ABB RAPID module: Module1.modx

MODULE Module1
    CONST robtarget Target_10:=[[355.425625842,0,585],[0.5,0,0.866025404,0],[0,0,0,0],[9E+09,9E+09,9E+09,9E+09,9E+09,9E+09]];
    CONST robtarget Target_20:=[[210.419326539,-286.445601335,585],[0.44609706,0.391142223,0.772662773,-0.225826068],[-1,-1,-1,0],[9E+09,9E+09,9E+09,9E+09,9E+09,9E+09]];

    CONST jointtarget JointTarget_0:=[[179.42,0.01,0.61,-29.68,-1.17,209.68],[9E+09,9E+09,9E+09,9E+09,9E+09,9E+09]];
    CONST jointtarget JointTarget_1:=[[178.84,0.03,1.21,-35.31,-2.01,215.3],[9E+09,9E+09,9E+09,9E+09,9E+09,9E+09]];
    CONST jointtarget JointTarget_2:=[[178.26,0.07,1.79,-37.62,-2.86,217.6],[9E+09,9E+09,9E+09,9E+09,9E+09,9E+09]];
    CONST jointtarget JointTarget_3:=[[177.68,0.12,2.37,-38.88,-3.7,218.83],[9E+09,9E+09,9E+09,9E+09,9E+09,9E+09]];
    CONST jointtarget JointTarget_4:=[[177.1,0.18,2.92,-39.66,-4.55,219.59],[9E+09,9E+09,9E+09,9E+09,9E+09,9E+09]];
    CONST jointtarget JointTarget_5:=[[176.52,0.26,3.47,-40.2,-5.4,220.1],[9E+09,9E+09,9E+09,9E+09,9E+09,9E+09]];
    CONST jointtarget JointTarget_6:=[[175.94,0.35,4.01,-40.6,-6.24,220.46],[9E+09,9E+09,9E+09,9E+09,9E+09,9E+09]];
    CONST jointtarget JointTarget_7:=[[175.36,0.45,4.53,-40.9,-7.09,220.71],[9E+09,9E+09,9E+09,9E+09,9E+09,9E+09]];
    CONST jointtarget JointTarget_8:=[[174.79,0.56,5.03,-41.13,-7.94,220.9],[9E+09,9E+09,9E+09,9E+09,9E+09,9E+09]];
    CONST jointtarget JointTarget_9:=[[174.21,0.69,5.53,-41.33,-8.78,221.03],[9E+09,9E+09,9E+09,9E+09,9E+09,9E+09]];
    CONST jointtarget JointTarget_10:=[[173.64,0.83,6.01,-41.49,-9.63,221.13],[9E+09,9E+09,9E+09,9E+09,9E+09,9E+09]];
    CONST jointtarget JointTarget_11:=[[173.07,0.98,6.48,-41.62,-10.47,221.19],[9E+09,9E+09,9E+09,9E+09,9E+09,9E+09]];
    CONST jointtarget JointTarget_12:=[[172.49,1.15,6.94,-41.74,-11.31,221.24],[9E+09,9E+09,9E+09,9E+09,9E+09,9E+09]];
    CONST jointtarget JointTarget_13:=[[171.93,1.33,7.38,-41.84,-12.15,221.26],[9E+09,9E+09,9E+09,9E+09,9E+09,9E+09]];
    CONST jointtarget JointTarget_14:=[[171.36,1.52,7.82,-41.94,-12.99,221.26],[9E+09,9E+09,9E+09,9E+09,9E+09,9E+09]];
    CONST jointtarget JointTarget_15:=[[170.79,1.73,8.23,-42.02,-13.83,221.25],[9E+09,9E+09,9E+09,9E+09,9E+09,9E+09]];
    CONST jointtarget JointTarget_16:=[[170.23,1.94,8.64,-42.1,-14.67,221.22],[9E+09,9E+09,9E+09,9E+09,9E+09,9E+09]];
    CONST jointtarget JointTarget_17:=[[169.67,2.17,9.03,-42.17,-15.5,221.19],[9E+09,9E+09,9E+09,9E+09,9E+09,9E+09]];
    CONST jointtarget JointTarget_18:=[[169.11,2.42,9.42,-42.24,-16.33,221.14],[9E+09,9E+09,9E+09,9E+09,9E+09,9E+09]];
    CONST jointtarget JointTarget_19:=[[168.55,2.67,9.78,-42.3,-17.16,221.09],[9E+09,9E+09,9E+09,9E+09,9E+09,9E+09]];
    CONST jointtarget JointTarget_20:=[[167.99,2.94,10.14,-42.36,-17.99,221.02],[9E+09,9E+09,9E+09,9E+09,9E+09,9E+09]];
    CONST jointtarget JointTarget_21:=[[167.44,3.22,10.48,-42.42,-18.81,220.95],[9E+09,9E+09,9E+09,9E+09,9E+09,9E+09]];
    CONST jointtarget JointTarget_22:=[[166.89,3.52,10.81,-42.48,-19.63,220.87],[9E+09,9E+09,9E+09,9E+09,9E+09,9E+09]];
    CONST jointtarget JointTarget_23:=[[166.34,3.82,11.13,-42.54,-20.45,220.78],[9E+09,9E+09,9E+09,9E+09,9E+09,9E+09]];
    CONST jointtarget JointTarget_24:=[[165.79,4.14,11.43,-42.6,-21.26,220.69],[9E+09,9E+09,9E+09,9E+09,9E+09,9E+09]];
    CONST jointtarget JointTarget_25:=[[165.25,4.47,11.72,-42.65,-22.07,220.6],[9E+09,9E+09,9E+09,9E+09,9E+09,9E+09]];
    CONST jointtarget JointTarget_26:=[[164.71,4.82,12,-42.71,-22.88,220.49],[9E+09,9E+09,9E+09,9E+09,9E+09,9E+09]];
    CONST jointtarget JointTarget_27:=[[164.17,5.17,12.26,-42.77,-23.68,220.38],[9E+09,9E+09,9E+09,9E+09,9E+09,9E+09]];
    CONST jointtarget JointTarget_28:=[[163.64,5.54,12.51,-42.83,-24.48,220.27],[9E+09,9E+09,9E+09,9E+09,9E+09,9E+09]];
    CONST jointtarget JointTarget_29:=[[163.11,5.91,12.75,-42.89,-25.27,220.16],[9E+09,9E+09,9E+09,9E+09,9E+09,9E+09]];
    CONST jointtarget JointTarget_30:=[[162.58,6.3,12.97,-42.96,-26.06,220.03],[9E+09,9E+09,9E+09,9E+09,9E+09,9E+09]];
    CONST jointtarget JointTarget_31:=[[162.05,6.7,13.19,-43.02,-26.85,219.91],[9E+09,9E+09,9E+09,9E+09,9E+09,9E+09]];
    CONST jointtarget JointTarget_32:=[[161.53,7.12,13.38,-43.09,-27.63,219.78],[9E+09,9E+09,9E+09,9E+09,9E+09,9E+09]];
    CONST jointtarget JointTarget_33:=[[161.01,7.54,13.57,-43.16,-28.41,219.65],[9E+09,9E+09,9E+09,9E+09,9E+09,9E+09]];
    CONST jointtarget JointTarget_34:=[[160.49,7.97,13.74,-43.23,-29.18,219.52],[9E+09,9E+09,9E+09,9E+09,9E+09,9E+09]];
    CONST jointtarget JointTarget_35:=[[159.98,8.42,13.9,-43.3,-29.94,219.38],[9E+09,9E+09,9E+09,9E+09,9E+09,9E+09]];
    CONST jointtarget JointTarget_36:=[[159.47,8.88,14.04,-43.37,-30.7,219.24],[9E+09,9E+09,9E+09,9E+09,9E+09,9E+09]];
    CONST jointtarget JointTarget_37:=[[158.97,9.34,14.18,-43.45,-31.46,219.1],[9E+09,9E+09,9E+09,9E+09,9E+09,9E+09]];
    CONST jointtarget JointTarget_38:=[[158.47,9.82,14.29,-43.53,-32.2,218.95],[9E+09,9E+09,9E+09,9E+09,9E+09,9E+09]];
    CONST jointtarget JointTarget_39:=[[157.97,10.31,14.4,-43.61,-32.94,218.81],[9E+09,9E+09,9E+09,9E+09,9E+09,9E+09]];
    CONST jointtarget JointTarget_40:=[[157.47,10.8,14.49,-43.7,-33.68,218.66],[9E+09,9E+09,9E+09,9E+09,9E+09,9E+09]];
    CONST jointtarget JointTarget_41:=[[156.98,11.31,14.57,-43.79,-34.41,218.51],[9E+09,9E+09,9E+09,9E+09,9E+09,9E+09]];
    CONST jointtarget JointTarget_42:=[[156.49,11.83,14.63,-43.88,-35.13,218.36],[9E+09,9E+09,9E+09,9E+09,9E+09,9E+09]];
    CONST jointtarget JointTarget_43:=[[156.01,12.35,14.68,-43.97,-35.85,218.2],[9E+09,9E+09,9E+09,9E+09,9E+09,9E+09]];
    CONST jointtarget JointTarget_44:=[[155.53,12.89,14.72,-44.07,-36.55,218.05],[9E+09,9E+09,9E+09,9E+09,9E+09,9E+09]];
    CONST jointtarget JointTarget_45:=[[155.05,13.43,14.74,-44.17,-37.25,217.9],[9E+09,9E+09,9E+09,9E+09,9E+09,9E+09]];
    CONST jointtarget JointTarget_46:=[[154.58,13.98,14.76,-44.27,-37.95,217.74],[9E+09,9E+09,9E+09,9E+09,9E+09,9E+09]];
    CONST jointtarget JointTarget_47:=[[154.11,14.54,14.75,-44.38,-38.63,217.59],[9E+09,9E+09,9E+09,9E+09,9E+09,9E+09]];
    CONST jointtarget JointTarget_48:=[[153.64,15.11,14.74,-44.49,-39.31,217.43],[9E+09,9E+09,9E+09,9E+09,9E+09,9E+09]];
    CONST jointtarget JointTarget_49:=[[153.18,15.69,14.71,-44.6,-39.98,217.28],[9E+09,9E+09,9E+09,9E+09,9E+09,9E+09]];
    CONST jointtarget JointTarget_50:=[[153.87,15.35,15.18,-43.63,-39.67,216.46],[9E+09,9E+09,9E+09,9E+09,9E+09,9E+09]];
    CONST jointtarget JointTarget_51:=[[154.56,15.02,15.64,-42.64,-39.35,215.64],[9E+09,9E+09,9E+09,9E+09,9E+09,9E+09]];
    CONST jointtarget JointTarget_52:=[[155.26,14.7,16.09,-41.63,-39.04,214.8],[9E+09,9E+09,9E+09,9E+09,9E+09,9E+09]];
    CONST jointtarget JointTarget_53:=[[155.98,14.38,16.52,-40.59,-38.73,213.94],[9E+09,9E+09,9E+09,9E+09,9E+09,9E+09]];
    CONST jointtarget JointTarget_54:=[[156.69,14.08,16.94,-39.54,-38.42,213.06],[9E+09,9E+09,9E+09,9E+09,9E+09,9E+09]];
    CONST jointtarget JointTarget_55:=[[157.42,13.78,17.35,-38.46,-38.12,212.17],[9E+09,9E+09,9E+09,9E+09,9E+09,9E+09]];
    CONST jointtarget JointTarget_56:=[[158.16,13.5,17.74,-37.36,-37.82,211.26],[9E+09,9E+09,9E+09,9E+09,9E+09,9E+09]];
    CONST jointtarget JointTarget_57:=[[158.9,13.22,18.12,-36.24,-37.52,210.32],[9E+09,9E+09,9E+09,9E+09,9E+09,9E+09]];
    CONST jointtarget JointTarget_58:=[[159.65,12.95,18.49,-35.09,-37.23,209.37],[9E+09,9E+09,9E+09,9E+09,9E+09,9E+09]];
    CONST jointtarget JointTarget_59:=[[160.41,12.69,18.85,-33.92,-36.94,208.4],[9E+09,9E+09,9E+09,9E+09,9E+09,9E+09]];
    CONST jointtarget JointTarget_60:=[[161.17,12.45,19.19,-32.72,-36.66,207.4],[9E+09,9E+09,9E+09,9E+09,9E+09,9E+09]];
    CONST jointtarget JointTarget_61:=[[161.94,12.21,19.52,-31.5,-36.39,206.39],[9E+09,9E+09,9E+09,9E+09,9E+09,9E+09]];
    CONST jointtarget JointTarget_62:=[[162.72,11.98,19.83,-30.26,-36.12,205.36],[9E+09,9E+09,9E+09,9E+09,9E+09,9E+09]];
    CONST jointtarget JointTarget_63:=[[163.5,11.76,20.13,-28.99,-35.86,204.3],[9E+09,9E+09,9E+09,9E+09,9E+09,9E+09]];
    CONST jointtarget JointTarget_64:=[[164.29,11.55,20.42,-27.7,-35.62,203.22],[9E+09,9E+09,9E+09,9E+09,9E+09,9E+09]];
    CONST jointtarget JointTarget_65:=[[165.09,11.36,20.69,-26.38,-35.38,202.13],[9E+09,9E+09,9E+09,9E+09,9E+09,9E+09]];
    CONST jointtarget JointTarget_66:=[[165.9,11.17,20.95,-25.04,-35.15,201.01],[9E+09,9E+09,9E+09,9E+09,9E+09,9E+09]];
    CONST jointtarget JointTarget_67:=[[166.7,11,21.19,-23.68,-34.93,199.87],[9E+09,9E+09,9E+09,9E+09,9E+09,9E+09]];
    CONST jointtarget JointTarget_68:=[[167.52,10.83,21.43,-22.3,-34.72,198.72],[9E+09,9E+09,9E+09,9E+09,9E+09,9E+09]];
    CONST jointtarget JointTarget_69:=[[168.34,10.68,21.64,-20.89,-34.53,197.54],[9E+09,9E+09,9E+09,9E+09,9E+09,9E+09]];
    CONST jointtarget JointTarget_70:=[[169.16,10.54,21.85,-19.47,-34.34,196.35],[9E+09,9E+09,9E+09,9E+09,9E+09,9E+09]];
    CONST jointtarget JointTarget_71:=[[169.99,10.41,22.04,-18.02,-34.17,195.14],[9E+09,9E+09,9E+09,9E+09,9E+09,9E+09]];
    CONST jointtarget JointTarget_72:=[[170.83,10.29,22.21,-16.56,-34.02,193.91],[9E+09,9E+09,9E+09,9E+09,9E+09,9E+09]];
    CONST jointtarget JointTarget_73:=[[171.66,10.18,22.37,-15.08,-33.88,192.67],[9E+09,9E+09,9E+09,9E+09,9E+09,9E+09]];
    CONST jointtarget JointTarget_74:=[[172.5,10.08,22.52,-13.58,-33.75,191.41],[9E+09,9E+09,9E+09,9E+09,9E+09,9E+09]];
    CONST jointtarget JointTarget_75:=[[173.35,10,22.65,-12.07,-33.64,190.14],[9E+09,9E+09,9E+09,9E+09,9E+09,9E+09]];
    CONST jointtarget JointTarget_76:=[[174.19,9.93,22.77,-10.55,-33.55,188.86],[9E+09,9E+09,9E+09,9E+09,9E+09,9E+09]];
    CONST jointtarget JointTarget_77:=[[175.04,9.87,22.87,-9.01,-33.47,187.57],[9E+09,9E+09,9E+09,9E+09,9E+09,9E+09]];
    CONST jointtarget JointTarget_78:=[[175.9,9.82,22.96,-7.47,-33.41,186.27],[9E+09,9E+09,9E+09,9E+09,9E+09,9E+09]];
    CONST jointtarget JointTarget_79:=[[176.75,9.79,23.04,-5.92,-33.36,184.97],[9E+09,9E+09,9E+09,9E+09,9E+09,9E+09]];
    CONST jointtarget JointTarget_80:=[[177.6,9.76,23.1,-4.36,-33.33,183.66],[9E+09,9E+09,9E+09,9E+09,9E+09,9E+09]];
    CONST jointtarget JointTarget_81:=[[178.46,9.75,23.14,-2.8,-33.32,182.35],[9E+09,9E+09,9E+09,9E+09,9E+09,9E+09]];
    CONST jointtarget JointTarget_82:=[[179.32,9.75,23.17,-1.24,-33.33,181.04],[9E+09,9E+09,9E+09,9E+09,9E+09,9E+09]];
    CONST jointtarget JointTarget_83:=[[180.17,9.76,23.19,0.32,-33.35,179.73],[9E+09,9E+09,9E+09,9E+09,9E+09,9E+09]];
    CONST jointtarget JointTarget_84:=[[181.03,9.79,23.19,1.87,-33.39,178.43],[9E+09,9E+09,9E+09,9E+09,9E+09,9E+09]];
    CONST jointtarget JointTarget_85:=[[181.89,9.83,23.18,3.43,-33.45,177.13],[9E+09,9E+09,9E+09,9E+09,9E+09,9E+09]];
    CONST jointtarget JointTarget_86:=[[182.74,9.88,23.15,4.97,-33.53,175.83],[9E+09,9E+09,9E+09,9E+09,9E+09,9E+09]];
    CONST jointtarget JointTarget_87:=[[183.6,9.94,23.11,6.51,-33.62,174.55],[9E+09,9E+09,9E+09,9E+09,9E+09,9E+09]];
    CONST jointtarget JointTarget_88:=[[184.45,10.01,23.06,8.03,-33.73,173.27],[9E+09,9E+09,9E+09,9E+09,9E+09,9E+09]];
    CONST jointtarget JointTarget_89:=[[185.3,10.1,22.98,9.55,-33.85,172.01],[9E+09,9E+09,9E+09,9E+09,9E+09,9E+09]];
    CONST jointtarget JointTarget_90:=[[186.15,10.19,22.9,11.05,-33.99,170.76],[9E+09,9E+09,9E+09,9E+09,9E+09,9E+09]];
    CONST jointtarget JointTarget_91:=[[187,10.3,22.8,12.53,-34.14,169.53],[9E+09,9E+09,9E+09,9E+09,9E+09,9E+09]];
    CONST jointtarget JointTarget_92:=[[187.84,10.42,22.69,14,-34.31,168.31],[9E+09,9E+09,9E+09,9E+09,9E+09,9E+09]];
    CONST jointtarget JointTarget_93:=[[188.68,10.55,22.56,15.45,-34.49,167.11],[9E+09,9E+09,9E+09,9E+09,9E+09,9E+09]];
    CONST jointtarget JointTarget_94:=[[189.51,10.7,22.42,16.88,-34.69,165.92],[9E+09,9E+09,9E+09,9E+09,9E+09,9E+09]];
    CONST jointtarget JointTarget_95:=[[190.34,10.85,22.26,18.29,-34.9,164.76],[9E+09,9E+09,9E+09,9E+09,9E+09,9E+09]];
    CONST jointtarget JointTarget_96:=[[191.17,11.02,22.09,19.68,-35.12,163.61],[9E+09,9E+09,9E+09,9E+09,9E+09,9E+09]];
    CONST jointtarget JointTarget_97:=[[191.99,11.2,21.9,21.05,-35.35,162.49],[9E+09,9E+09,9E+09,9E+09,9E+09,9E+09]];
    CONST jointtarget JointTarget_98:=[[192.81,11.39,21.7,22.39,-35.6,161.39],[9E+09,9E+09,9E+09,9E+09,9E+09,9E+09]];
    CONST jointtarget JointTarget_99:=[[193.62,11.59,21.49,23.71,-35.85,160.3],[9E+09,9E+09,9E+09,9E+09,9E+09,9E+09]];
    CONST jointtarget JointTarget_100:=[[193.15,11.97,21.97,22.48,-36.49,161.5],[9E+09,9E+09,9E+09,9E+09,9E+09,9E+09]];
    CONST jointtarget JointTarget_101:=[[192.67,12.37,22.44,21.3,-37.15,162.65],[9E+09,9E+09,9E+09,9E+09,9E+09,9E+09]];
    CONST jointtarget JointTarget_102:=[[192.19,12.79,22.89,20.15,-37.82,163.75],[9E+09,9E+09,9E+09,9E+09,9E+09,9E+09]];
    CONST jointtarget JointTarget_103:=[[191.71,13.22,23.33,19.03,-38.51,164.81],[9E+09,9E+09,9E+09,9E+09,9E+09,9E+09]];
    CONST jointtarget JointTarget_104:=[[191.23,13.67,23.75,17.95,-39.22,165.83],[9E+09,9E+09,9E+09,9E+09,9E+09,9E+09]];
    CONST jointtarget JointTarget_105:=[[190.75,14.14,24.15,16.9,-39.93,166.81],[9E+09,9E+09,9E+09,9E+09,9E+09,9E+09]];
    CONST jointtarget JointTarget_106:=[[190.27,14.62,24.54,15.88,-40.66,167.75],[9E+09,9E+09,9E+09,9E+09,9E+09,9E+09]];
    CONST jointtarget JointTarget_107:=[[189.78,15.12,24.91,14.89,-41.41,168.66],[9E+09,9E+09,9E+09,9E+09,9E+09,9E+09]];
    CONST jointtarget JointTarget_108:=[[189.3,15.64,25.26,13.93,-42.16,169.52],[9E+09,9E+09,9E+09,9E+09,9E+09,9E+09]];
    CONST jointtarget JointTarget_109:=[[188.81,16.18,25.6,12.99,-42.92,170.35],[9E+09,9E+09,9E+09,9E+09,9E+09,9E+09]];
    CONST jointtarget JointTarget_110:=[[188.32,16.73,25.92,12.09,-43.69,171.14],[9E+09,9E+09,9E+09,9E+09,9E+09,9E+09]];
    CONST jointtarget JointTarget_111:=[[187.83,17.3,26.22,11.21,-44.47,171.9],[9E+09,9E+09,9E+09,9E+09,9E+09,9E+09]];
    CONST jointtarget JointTarget_112:=[[187.34,17.88,26.51,10.36,-45.26,172.62],[9E+09,9E+09,9E+09,9E+09,9E+09,9E+09]];
    CONST jointtarget JointTarget_113:=[[186.84,18.48,26.78,9.53,-46.06,173.31],[9E+09,9E+09,9E+09,9E+09,9E+09,9E+09]];
    CONST jointtarget JointTarget_114:=[[186.35,19.09,27.03,8.72,-46.86,173.97],[9E+09,9E+09,9E+09,9E+09,9E+09,9E+09]];
    CONST jointtarget JointTarget_115:=[[185.86,19.72,27.27,7.93,-47.66,174.6],[9E+09,9E+09,9E+09,9E+09,9E+09,9E+09]];
    CONST jointtarget JointTarget_116:=[[185.36,20.37,27.48,7.17,-48.47,175.2],[9E+09,9E+09,9E+09,9E+09,9E+09,9E+09]];
    CONST jointtarget JointTarget_117:=[[184.86,21.02,27.68,6.42,-49.29,175.77],[9E+09,9E+09,9E+09,9E+09,9E+09,9E+09]];
    CONST jointtarget JointTarget_118:=[[184.37,21.7,27.87,5.7,-50.1,176.31],[9E+09,9E+09,9E+09,9E+09,9E+09,9E+09]];
    CONST jointtarget JointTarget_119:=[[183.87,22.38,28.03,4.99,-50.92,176.82],[9E+09,9E+09,9E+09,9E+09,9E+09,9E+09]];
    CONST jointtarget JointTarget_120:=[[183.37,23.09,28.18,4.29,-51.74,177.31],[9E+09,9E+09,9E+09,9E+09,9E+09,9E+09]];
    CONST jointtarget JointTarget_121:=[[182.87,23.8,28.3,3.62,-52.56,177.78],[9E+09,9E+09,9E+09,9E+09,9E+09,9E+09]];
    CONST jointtarget JointTarget_122:=[[182.37,24.53,28.41,2.96,-53.37,178.22],[9E+09,9E+09,9E+09,9E+09,9E+09,9E+09]];
    CONST jointtarget JointTarget_123:=[[181.87,25.26,28.5,2.31,-54.19,178.64],[9E+09,9E+09,9E+09,9E+09,9E+09,9E+09]];
    CONST jointtarget JointTarget_124:=[[181.37,26.02,28.58,1.68,-55,179.03],[9E+09,9E+09,9E+09,9E+09,9E+09,9E+09]];
    CONST jointtarget JointTarget_125:=[[180.87,26.78,28.63,1.05,-55.81,179.4],[9E+09,9E+09,9E+09,9E+09,9E+09,9E+09]];
    CONST jointtarget JointTarget_126:=[[180.37,27.55,28.67,0.45,-56.62,179.75],[9E+09,9E+09,9E+09,9E+09,9E+09,9E+09]];
    CONST jointtarget JointTarget_127:=[[179.87,28.33,28.69,-0.15,-57.42,180.08],[9E+09,9E+09,9E+09,9E+09,9E+09,9E+09]];
    CONST jointtarget JointTarget_128:=[[179.37,29.13,28.69,-0.74,-58.22,180.39],[9E+09,9E+09,9E+09,9E+09,9E+09,9E+09]];
    CONST jointtarget JointTarget_129:=[[178.87,29.93,28.67,-1.32,-59.01,180.69],[9E+09,9E+09,9E+09,9E+09,9E+09,9E+09]];
    CONST jointtarget JointTarget_130:=[[178.37,30.74,28.64,-1.89,-59.79,180.96],[9E+09,9E+09,9E+09,9E+09,9E+09,9E+09]];
    CONST jointtarget JointTarget_131:=[[177.87,31.56,28.58,-2.44,-60.57,181.22],[9E+09,9E+09,9E+09,9E+09,9E+09,9E+09]];
    CONST jointtarget JointTarget_132:=[[177.37,32.39,28.51,-3,-61.34,181.46],[9E+09,9E+09,9E+09,9E+09,9E+09,9E+09]];
    CONST jointtarget JointTarget_133:=[[176.87,33.23,28.42,-3.54,-62.09,181.68],[9E+09,9E+09,9E+09,9E+09,9E+09,9E+09]];
    CONST jointtarget JointTarget_134:=[[176.37,34.07,28.31,-4.08,-62.84,181.89],[9E+09,9E+09,9E+09,9E+09,9E+09,9E+09]];
    CONST jointtarget JointTarget_135:=[[175.88,34.92,28.19,-4.61,-63.58,182.08],[9E+09,9E+09,9E+09,9E+09,9E+09,9E+09]];
    CONST jointtarget JointTarget_136:=[[175.38,35.78,28.04,-5.13,-64.31,182.26],[9E+09,9E+09,9E+09,9E+09,9E+09,9E+09]];
    CONST jointtarget JointTarget_137:=[[174.88,36.64,27.88,-5.65,-65.03,182.43],[9E+09,9E+09,9E+09,9E+09,9E+09,9E+09]];
    CONST jointtarget JointTarget_138:=[[174.39,37.5,27.7,-6.16,-65.73,182.58],[9E+09,9E+09,9E+09,9E+09,9E+09,9E+09]];
    CONST jointtarget JointTarget_139:=[[173.89,38.37,27.5,-6.67,-66.42,182.72],[9E+09,9E+09,9E+09,9E+09,9E+09,9E+09]];
    CONST jointtarget JointTarget_140:=[[173.4,39.25,27.29,-7.17,-67.1,182.85],[9E+09,9E+09,9E+09,9E+09,9E+09,9E+09]];
    CONST jointtarget JointTarget_141:=[[172.9,40.13,27.05,-7.67,-67.77,182.97],[9E+09,9E+09,9E+09,9E+09,9E+09,9E+09]];
    CONST jointtarget JointTarget_142:=[[172.41,41.01,26.8,-8.17,-68.42,183.07],[9E+09,9E+09,9E+09,9E+09,9E+09,9E+09]];
    CONST jointtarget JointTarget_143:=[[171.92,41.9,26.54,-8.66,-69.06,183.17],[9E+09,9E+09,9E+09,9E+09,9E+09,9E+09]];
    CONST jointtarget JointTarget_144:=[[171.43,42.78,26.25,-9.14,-69.68,183.26],[9E+09,9E+09,9E+09,9E+09,9E+09,9E+09]];
    CONST jointtarget JointTarget_145:=[[170.94,43.67,25.95,-9.63,-70.29,183.34],[9E+09,9E+09,9E+09,9E+09,9E+09,9E+09]];
    CONST jointtarget JointTarget_146:=[[170.45,44.56,25.63,-10.11,-70.88,183.41],[9E+09,9E+09,9E+09,9E+09,9E+09,9E+09]];
    CONST jointtarget JointTarget_147:=[[169.97,45.46,25.29,-10.59,-71.46,183.47],[9E+09,9E+09,9E+09,9E+09,9E+09,9E+09]];
    CONST jointtarget JointTarget_148:=[[169.48,46.35,24.94,-11.06,-72.02,183.53],[9E+09,9E+09,9E+09,9E+09,9E+09,9E+09]];
    CONST jointtarget JointTarget_149:=[[169,47.25,24.57,-11.54,-72.56,183.58],[9E+09,9E+09,9E+09,9E+09,9E+09,9E+09]];


    PROC main()
        Path_10;
    ENDPROC
    PROC Path_10()
        !MoveL Target_10,v1000,z100,tool0\WObj:=wobj0;
        !MoveL Target_20,v1000,z100,tool0\WObj:=wobj0;

        MoveAbsJ JointTarget_0,v100,z1,tool0\WObj:=wobj0;
        MoveAbsJ JointTarget_1,v100,z1,tool0\WObj:=wobj0;
        MoveAbsJ JointTarget_2,v100,z1,tool0\WObj:=wobj0;
        MoveAbsJ JointTarget_3,v100,z1,tool0\WObj:=wobj0;
        MoveAbsJ JointTarget_4,v100,z1,tool0\WObj:=wobj0;
        MoveAbsJ JointTarget_5,v100,z1,tool0\WObj:=wobj0;
        MoveAbsJ JointTarget_6,v100,z1,tool0\WObj:=wobj0;
        MoveAbsJ JointTarget_7,v100,z1,tool0\WObj:=wobj0;
        MoveAbsJ JointTarget_8,v100,z1,tool0\WObj:=wobj0;
        MoveAbsJ JointTarget_9,v100,z1,tool0\WObj:=wobj0;
        MoveAbsJ JointTarget_10,v100,z1,tool0\WObj:=wobj0;
        MoveAbsJ JointTarget_11,v100,z1,tool0\WObj:=wobj0;
        MoveAbsJ JointTarget_12,v100,z1,tool0\WObj:=wobj0;
        MoveAbsJ JointTarget_13,v100,z1,tool0\WObj:=wobj0;
        MoveAbsJ JointTarget_14,v100,z1,tool0\WObj:=wobj0;
        MoveAbsJ JointTarget_15,v100,z1,tool0\WObj:=wobj0;
        MoveAbsJ JointTarget_16,v100,z1,tool0\WObj:=wobj0;
        MoveAbsJ JointTarget_17,v100,z1,tool0\WObj:=wobj0;
        MoveAbsJ JointTarget_18,v100,z1,tool0\WObj:=wobj0;
        MoveAbsJ JointTarget_19,v100,z1,tool0\WObj:=wobj0;
        MoveAbsJ JointTarget_20,v100,z1,tool0\WObj:=wobj0;
        MoveAbsJ JointTarget_21,v100,z1,tool0\WObj:=wobj0;
        MoveAbsJ JointTarget_22,v100,z1,tool0\WObj:=wobj0;
        MoveAbsJ JointTarget_23,v100,z1,tool0\WObj:=wobj0;
        MoveAbsJ JointTarget_24,v100,z1,tool0\WObj:=wobj0;
        MoveAbsJ JointTarget_25,v100,z1,tool0\WObj:=wobj0;
        MoveAbsJ JointTarget_26,v100,z1,tool0\WObj:=wobj0;
        MoveAbsJ JointTarget_27,v100,z1,tool0\WObj:=wobj0;
        MoveAbsJ JointTarget_28,v100,z1,tool0\WObj:=wobj0;
        MoveAbsJ JointTarget_29,v100,z1,tool0\WObj:=wobj0;
        MoveAbsJ JointTarget_30,v100,z1,tool0\WObj:=wobj0;
        MoveAbsJ JointTarget_31,v100,z1,tool0\WObj:=wobj0;
        MoveAbsJ JointTarget_32,v100,z1,tool0\WObj:=wobj0;
        MoveAbsJ JointTarget_33,v100,z1,tool0\WObj:=wobj0;
        MoveAbsJ JointTarget_34,v100,z1,tool0\WObj:=wobj0;
        MoveAbsJ JointTarget_35,v100,z1,tool0\WObj:=wobj0;
        MoveAbsJ JointTarget_36,v100,z1,tool0\WObj:=wobj0;
        MoveAbsJ JointTarget_37,v100,z1,tool0\WObj:=wobj0;
        MoveAbsJ JointTarget_38,v100,z1,tool0\WObj:=wobj0;
        MoveAbsJ JointTarget_39,v100,z1,tool0\WObj:=wobj0;
        MoveAbsJ JointTarget_40,v100,z1,tool0\WObj:=wobj0;
        MoveAbsJ JointTarget_41,v100,z1,tool0\WObj:=wobj0;
        MoveAbsJ JointTarget_42,v100,z1,tool0\WObj:=wobj0;
        MoveAbsJ JointTarget_43,v100,z1,tool0\WObj:=wobj0;
        MoveAbsJ JointTarget_44,v100,z1,tool0\WObj:=wobj0;
        MoveAbsJ JointTarget_45,v100,z1,tool0\WObj:=wobj0;
        MoveAbsJ JointTarget_46,v100,z1,tool0\WObj:=wobj0;
        MoveAbsJ JointTarget_47,v100,z1,tool0\WObj:=wobj0;
        MoveAbsJ JointTarget_48,v100,z1,tool0\WObj:=wobj0;
        MoveAbsJ JointTarget_49,v100,z1,tool0\WObj:=wobj0;
        MoveAbsJ JointTarget_50,v100,z1,tool0\WObj:=wobj0;
        MoveAbsJ JointTarget_51,v100,z1,tool0\WObj:=wobj0;
        MoveAbsJ JointTarget_52,v100,z1,tool0\WObj:=wobj0;
        MoveAbsJ JointTarget_53,v100,z1,tool0\WObj:=wobj0;
        MoveAbsJ JointTarget_54,v100,z1,tool0\WObj:=wobj0;
        MoveAbsJ JointTarget_55,v100,z1,tool0\WObj:=wobj0;
        MoveAbsJ JointTarget_56,v100,z1,tool0\WObj:=wobj0;
        MoveAbsJ JointTarget_57,v100,z1,tool0\WObj:=wobj0;
        MoveAbsJ JointTarget_58,v100,z1,tool0\WObj:=wobj0;
        MoveAbsJ JointTarget_59,v100,z1,tool0\WObj:=wobj0;
        MoveAbsJ JointTarget_60,v100,z1,tool0\WObj:=wobj0;
        MoveAbsJ JointTarget_61,v100,z1,tool0\WObj:=wobj0;
        MoveAbsJ JointTarget_62,v100,z1,tool0\WObj:=wobj0;
        MoveAbsJ JointTarget_63,v100,z1,tool0\WObj:=wobj0;
        MoveAbsJ JointTarget_64,v100,z1,tool0\WObj:=wobj0;
        MoveAbsJ JointTarget_65,v100,z1,tool0\WObj:=wobj0;
        MoveAbsJ JointTarget_66,v100,z1,tool0\WObj:=wobj0;
        MoveAbsJ JointTarget_67,v100,z1,tool0\WObj:=wobj0;
        MoveAbsJ JointTarget_68,v100,z1,tool0\WObj:=wobj0;
        MoveAbsJ JointTarget_69,v100,z1,tool0\WObj:=wobj0;
        MoveAbsJ JointTarget_70,v100,z1,tool0\WObj:=wobj0;
        MoveAbsJ JointTarget_71,v100,z1,tool0\WObj:=wobj0;
        MoveAbsJ JointTarget_72,v100,z1,tool0\WObj:=wobj0;
        MoveAbsJ JointTarget_73,v100,z1,tool0\WObj:=wobj0;
        MoveAbsJ JointTarget_74,v100,z1,tool0\WObj:=wobj0;
        MoveAbsJ JointTarget_75,v100,z1,tool0\WObj:=wobj0;
        MoveAbsJ JointTarget_76,v100,z1,tool0\WObj:=wobj0;
        MoveAbsJ JointTarget_77,v100,z1,tool0\WObj:=wobj0;
        MoveAbsJ JointTarget_78,v100,z1,tool0\WObj:=wobj0;
        MoveAbsJ JointTarget_79,v100,z1,tool0\WObj:=wobj0;
        MoveAbsJ JointTarget_80,v100,z1,tool0\WObj:=wobj0;
        MoveAbsJ JointTarget_81,v100,z1,tool0\WObj:=wobj0;
        MoveAbsJ JointTarget_82,v100,z1,tool0\WObj:=wobj0;
        MoveAbsJ JointTarget_83,v100,z1,tool0\WObj:=wobj0;
        MoveAbsJ JointTarget_84,v100,z1,tool0\WObj:=wobj0;
        MoveAbsJ JointTarget_85,v100,z1,tool0\WObj:=wobj0;
        MoveAbsJ JointTarget_86,v100,z1,tool0\WObj:=wobj0;
        MoveAbsJ JointTarget_87,v100,z1,tool0\WObj:=wobj0;
        MoveAbsJ JointTarget_88,v100,z1,tool0\WObj:=wobj0;
        MoveAbsJ JointTarget_89,v100,z1,tool0\WObj:=wobj0;
        MoveAbsJ JointTarget_90,v100,z1,tool0\WObj:=wobj0;
        MoveAbsJ JointTarget_91,v100,z1,tool0\WObj:=wobj0;
        MoveAbsJ JointTarget_92,v100,z1,tool0\WObj:=wobj0;
        MoveAbsJ JointTarget_93,v100,z1,tool0\WObj:=wobj0;
        MoveAbsJ JointTarget_94,v100,z1,tool0\WObj:=wobj0;
        MoveAbsJ JointTarget_95,v100,z1,tool0\WObj:=wobj0;
        MoveAbsJ JointTarget_96,v100,z1,tool0\WObj:=wobj0;
        MoveAbsJ JointTarget_97,v100,z1,tool0\WObj:=wobj0;
        MoveAbsJ JointTarget_98,v100,z1,tool0\WObj:=wobj0;
        MoveAbsJ JointTarget_99,v100,z1,tool0\WObj:=wobj0;
        MoveAbsJ JointTarget_100,v100,z1,tool0\WObj:=wobj0;
        MoveAbsJ JointTarget_101,v100,z1,tool0\WObj:=wobj0;
        MoveAbsJ JointTarget_102,v100,z1,tool0\WObj:=wobj0;
        MoveAbsJ JointTarget_103,v100,z1,tool0\WObj:=wobj0;
        MoveAbsJ JointTarget_104,v100,z1,tool0\WObj:=wobj0;
        MoveAbsJ JointTarget_105,v100,z1,tool0\WObj:=wobj0;
        MoveAbsJ JointTarget_106,v100,z1,tool0\WObj:=wobj0;
        MoveAbsJ JointTarget_107,v100,z1,tool0\WObj:=wobj0;
        MoveAbsJ JointTarget_108,v100,z1,tool0\WObj:=wobj0;
        MoveAbsJ JointTarget_109,v100,z1,tool0\WObj:=wobj0;
        MoveAbsJ JointTarget_110,v100,z1,tool0\WObj:=wobj0;
        MoveAbsJ JointTarget_111,v100,z1,tool0\WObj:=wobj0;
        MoveAbsJ JointTarget_112,v100,z1,tool0\WObj:=wobj0;
        MoveAbsJ JointTarget_113,v100,z1,tool0\WObj:=wobj0;
        MoveAbsJ JointTarget_114,v100,z1,tool0\WObj:=wobj0;
        MoveAbsJ JointTarget_115,v100,z1,tool0\WObj:=wobj0;
        MoveAbsJ JointTarget_116,v100,z1,tool0\WObj:=wobj0;
        MoveAbsJ JointTarget_117,v100,z1,tool0\WObj:=wobj0;
        MoveAbsJ JointTarget_118,v100,z1,tool0\WObj:=wobj0;
        MoveAbsJ JointTarget_119,v100,z1,tool0\WObj:=wobj0;
        MoveAbsJ JointTarget_120,v100,z1,tool0\WObj:=wobj0;
        MoveAbsJ JointTarget_121,v100,z1,tool0\WObj:=wobj0;
        MoveAbsJ JointTarget_122,v100,z1,tool0\WObj:=wobj0;
        MoveAbsJ JointTarget_123,v100,z1,tool0\WObj:=wobj0;
        MoveAbsJ JointTarget_124,v100,z1,tool0\WObj:=wobj0;
        MoveAbsJ JointTarget_125,v100,z1,tool0\WObj:=wobj0;
        MoveAbsJ JointTarget_126,v100,z1,tool0\WObj:=wobj0;
        MoveAbsJ JointTarget_127,v100,z1,tool0\WObj:=wobj0;
        MoveAbsJ JointTarget_128,v100,z1,tool0\WObj:=wobj0;
        MoveAbsJ JointTarget_129,v100,z1,tool0\WObj:=wobj0;
        MoveAbsJ JointTarget_130,v100,z1,tool0\WObj:=wobj0;
        MoveAbsJ JointTarget_131,v100,z1,tool0\WObj:=wobj0;
        MoveAbsJ JointTarget_132,v100,z1,tool0\WObj:=wobj0;
        MoveAbsJ JointTarget_133,v100,z1,tool0\WObj:=wobj0;
        MoveAbsJ JointTarget_134,v100,z1,tool0\WObj:=wobj0;
        MoveAbsJ JointTarget_135,v100,z1,tool0\WObj:=wobj0;
        MoveAbsJ JointTarget_136,v100,z1,tool0\WObj:=wobj0;
        MoveAbsJ JointTarget_137,v100,z1,tool0\WObj:=wobj0;
        MoveAbsJ JointTarget_138,v100,z1,tool0\WObj:=wobj0;
        MoveAbsJ JointTarget_139,v100,z1,tool0\WObj:=wobj0;
        MoveAbsJ JointTarget_140,v100,z1,tool0\WObj:=wobj0;
        MoveAbsJ JointTarget_141,v100,z1,tool0\WObj:=wobj0;
        MoveAbsJ JointTarget_142,v100,z1,tool0\WObj:=wobj0;
        MoveAbsJ JointTarget_143,v100,z1,tool0\WObj:=wobj0;
        MoveAbsJ JointTarget_144,v100,z1,tool0\WObj:=wobj0;
        MoveAbsJ JointTarget_145,v100,z1,tool0\WObj:=wobj0;
        MoveAbsJ JointTarget_146,v100,z1,tool0\WObj:=wobj0;
        MoveAbsJ JointTarget_147,v100,z1,tool0\WObj:=wobj0;
        MoveAbsJ JointTarget_148,v100,z1,tool0\WObj:=wobj0;
        MoveAbsJ JointTarget_149,v100,z1,tool0\WObj:=wobj0;
    ENDPROC
ENDMODULE
